(**
This function block abstracts the Beckhoff EtherCAT terminal EL2624
*)
FUNCTION_BLOCK EL2624 IMPLEMENTS I_terminal_execution
VAR_INPUT
END_VAR
VAR_OUTPUT
	DO_channel_1 		: I_HAL_DO :=_channel_1;
	DO_channel_2 		: I_HAL_DO :=_channel_2;
	DO_channel_3 		: I_HAL_DO :=_channel_3;
	DO_channel_4 		: I_HAL_DO :=_channel_4;
END_VAR
VAR
	WcState_WcState			AT%I*: BOOL;
	InfoData_State			AT%I*: UINT;
	
	Channel_1_Output         AT%Q*: BOOL;
	Channel_2_Output         AT%Q*: BOOL;
	Channel_3_Output         AT%Q*: BOOL;
	Channel_4_Output         AT%Q*: BOOL;
	
	_channel_1 : HAL_DO_Channel(channel_number:=1);
	_channel_2 : HAL_DO_Channel(channel_number:=2);
	_channel_3 : HAL_DO_Channel(channel_number:=3);
	_channel_4 : HAL_DO_Channel(channel_number:=4);
END_VAR
VAR CONSTANT	
    HARDWARE_REVSION : UINT:=19;
END_VAR


_channel_1.wcState:= NOT  WcState_WcState;
_channel_2.wcState:= NOT  WcState_WcState;
_channel_3.wcState:= NOT  WcState_WcState;
_channel_4.wcState:= NOT  WcState_WcState;

_channel_1();
_channel_2();
_channel_3();
_channel_4();

Channel_1_Output := _channel_1.terminal_value;
Channel_2_Output := _channel_2.terminal_value;
Channel_3_Output := _channel_3.terminal_value;
Channel_4_Output := _channel_4.terminal_value;

METHOD FB_init : BOOL
VAR_INPUT
	bInitRetains : BOOL; // if TRUE, the retain variables are initialized (warm start / cold start)
	bInCopyCode : BOOL;  // if TRUE, the instance afterwards gets moved into the copy code (online change)
	CoE_communication_handler : I_CoE_communication_handler;
END_VAR
END_METHOD

METHOD run : BOOL
VAR_INPUT
END_VAR
THIS^();
END_METHOD

END_FUNCTION_BLOCK

(* stored: Version 1.1.0.1, ProductVersion 3.1.4024.6
   POU EL2624: Id {ce1f63ab-fafb-0d1e-06a6-c0b9d6a1eb20}, SpecialFunc None
   Method FB_init: Id {f58d1963-c27a-055b-3ca6-2beb0221c335}
   Method run: Id {5339e4c4-de24-0ad6-27cc-d3ca3ceb6a9a} *)
